FUNCTION_BLOCK FB_LensSet_Test EXTENDS FB_TestSuiteExtended


TestIndexIndexInRangeExpectTrue();

TestSetInvalidNumLensesExpectErrorNoChangeToValue();

TestSetLensGetLensExpectNoErrorCorrectValue();

TestSetNumLensesGetNumLensesExpectNoErrorValueSet();

TestTooHighIndexIndexInRangeExpectFalse();

TestTooLowIndexIndexInRangeExpectFalse();


METHOD TestIndexIndexInRangeExpectTrue
VAR
    // Subject under test
    fbLensSet : FB_LensSet;
    bResult : BOOL;
END_VAR

TEST('TestIndexIndexInRangeExpectTrue');

// Test Fixture
fbLensSet.NumLenses:= 9;

// Here the test starts
bResult := fbLensSet.IndexInRange(nIndex := 9);

AssertNoError(Fallible := fbLensSet);

AssertTrue(
    Condition := bResult,
    Message := 'Index should have registered as in range.'
);

TEST_FINISHED();
END_METHOD


METHOD TestSetInvalidNumLensesExpectErrorNoChangeToValue
VAR
    // Subject under test
    fbLensSet : FB_LensSet;
    nNumLenses : INT;
END_VAR

TEST('TestSetInvalidNumLensesExpectErrorNoChangeToValue');

// Test Fixture
nNumLenses := 5;
fbLensSet.NumLenses:= nNumLenses;

// Here the test starts
fbLensSet.NumLenses := 0;

AssertError(Fallible := fbLensSet);

AssertEquals_INT(
    Expected := nNumLenses,
    Actual := fbLensSet.NumLenses,
    Message := 'NumLenses should not have changed.'
);

TEST_FINISHED();
END_METHOD


METHOD TestSetLensGetLensExpectNoErrorCorrectValue
VAR
    fbLensMock : FB_LensMock;
    fbRadiusMock : FB_QuantityLREALPublicMock;

    // Subject under test
    fbLensSet : FB_LensSet;
    fbLens : FB_Lens;
    fbRadiusResult : FB_QuantityLREALPublic(Units := 'm');

    sExpected : T_MaxString;
    nExpected : INT;
    sResult : T_MaxString;
    nResult : INT;
END_VAR

TEST('TestSetMaterialNameOfGetMaterialNameOfExpectNoErrorCorrectValue');

// Test Fixture
sExpected := 'Material1';
nExpected := 32;

fbRadiusMock.Val := 27.65;
fbRadiusMock.Units := 'cm';

fbLensSet.NumLenses:= 5;

fbLensMock.MaterialFormula := sExpected;
fbLensMock.Multiplier := nExpected;
fbLensMock.SetRadius(Radius := fbRadiusMock);

// Here the test starts
fbLensSet.SetLens(LensNum := 1, Lens := fbLensMock);
fbLensSet.GetLens(LensNum := 1, Lens := fbLens);

sResult := fbLens.MaterialFormula;
nResult := fbLens.Multiplier;
fbLens.GetRadius(Radius := fbRadiusResult);

AssertNoError(Fallible := fbLensSet);

AssertEquals_STRING(
    Expected := sExpected,
    Actual := sResult,
    Message := 'String did not have the correct value.'
);

AssertEquals_INT(
    Expected := nExpected,
    Actual := nResult,
    Message := 'Multiplier did not have the correct value.'
);

AssertNoErrorExactExpectedQuantityLREAL(
    Expected := fbRadiusMock,
    Actual := fbRadiusResult
);

TEST_FINISHED();
END_METHOD


METHOD TestSetNumLensesGetNumLensesExpectNoErrorValueSet
VAR
    fbConvertUnitsLREALMock : FB_ConvertUnitsLREALMock;
    fbCalcFocalLengthSingleLens : FB_CalcFocalLengthSingleLensMock;
    // Subject under test
    fbLensSet : FB_LensSet;
    nNumLenses : INT;
END_VAR

TEST('TestSetNumLensesGetNumLensesExpectNoErrorValueSet');

// Test Fixture
nNumLenses := 5;

// Here the test starts
fbLensSet.NumLenses:= nNumLenses;

AssertNoError(Fallible := fbLensSet);

AssertEquals_INT(
    Expected := nNumLenses,
    Actual := fbLensSet.NumLenses,
    Message := 'NumLenses did not set properly.'
);

TEST_FINISHED();
END_METHOD


METHOD TestTooHighIndexIndexInRangeExpectFalse
VAR
    // Subject under test
    fbLensSet : FB_LensSet;
    bResult : BOOL;
END_VAR

TEST('TestTooHighIndexIndexInRangeExpectFalse');

// Test Fixture
fbLensSet.NumLenses:= 9;

// Here the test starts
bResult := fbLensSet.IndexInRange(nIndex := fbLensSet.NumLenses + 1);

AssertNoError(Fallible := fbLensSet);

AssertFalse(
    Condition := bResult,
    Message := 'Index should have registered as out of range.'
);

TEST_FINISHED();
END_METHOD


METHOD TestTooLowIndexIndexInRangeExpectFalse
VAR
    // Subject under test
    fbLensSet : FB_LensSet;
    bResult : BOOL;
END_VAR

TEST('TestTooLowIndexIndexInRangeExpectFalse');

// Test Fixture
fbLensSet.NumLenses:= 9;

// Here the test starts
bResult := fbLensSet.IndexInRange(nIndex := 0);

AssertNoError(Fallible := fbLensSet);

AssertFalse(
    Condition := bResult,
    Message := 'Index should have registered as out of range.'
);

TEST_FINISHED();
END_METHOD

END_FUNCTION_BLOCK

(* stored: Version 1.1.0.1
   POU FB_LensSet_Test: Id {959fcf0e-1b33-40b1-a7be-9a4bd9a118a1}, SpecialFunc None
   Method TestIndexIndexInRangeExpectTrue: Id {1564fb33-badf-45fa-8b05-f60c5ace519e}
   Method TestSetInvalidNumLensesExpectErrorNoChangeToValue: Id {6e1a08f1-05bf-4a64-a3f2-0ce2e1fad65f}
   Method TestSetLensGetLensExpectNoErrorCorrectValue: Id {06da589f-bfc8-49ef-b9bc-1f973a59e2e8}
   Method TestSetNumLensesGetNumLensesExpectNoErrorValueSet: Id {bf018f87-a842-4889-8d85-6accaf0c30dd}
   Method TestTooHighIndexIndexInRangeExpectFalse: Id {af6a7413-9b4b-4008-b3a7-e0c356c39a51}
   Method TestTooLowIndexIndexInRangeExpectFalse: Id {0acb188b-4d74-41f8-aaf5-43b264bf17d3} *)
